% RSLogix 500 project Project6-Final.RSS, saved by version 8.30.00.16 %
PROJECT "UNTITLED"    % processor: Bul.1763 MicroLogix 1100 Series B %

PROGRAM FILES
  LAD 2 "MAIN"  2 rungs
  LAD 3 "LOGIC"  10 rungs

DATA FILES
  O0 OUTPUT  4 elements
  I1 INPUT  6 elements
  S2 STATUS  66 elements
  B3 BINARY  2 elements
  T4 TIMER  1 elements
  C5 COUNTER  4 elements
  R6 CONTROL  1 elements
  N7 INTEGER  4 elements
  F8 FLOAT  1 elements

LADDER 2 "MAIN"
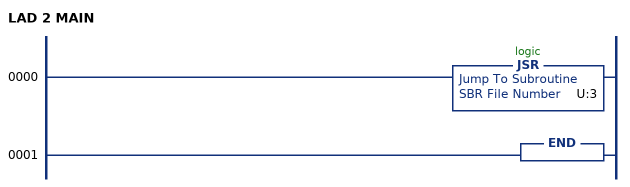
% Rung: 0 %
SOR JSR U:3 EOR
%   U:3  "logic" %
% Rung: 1 %
SOR END EOR

LADDER 3 "LOGIC"
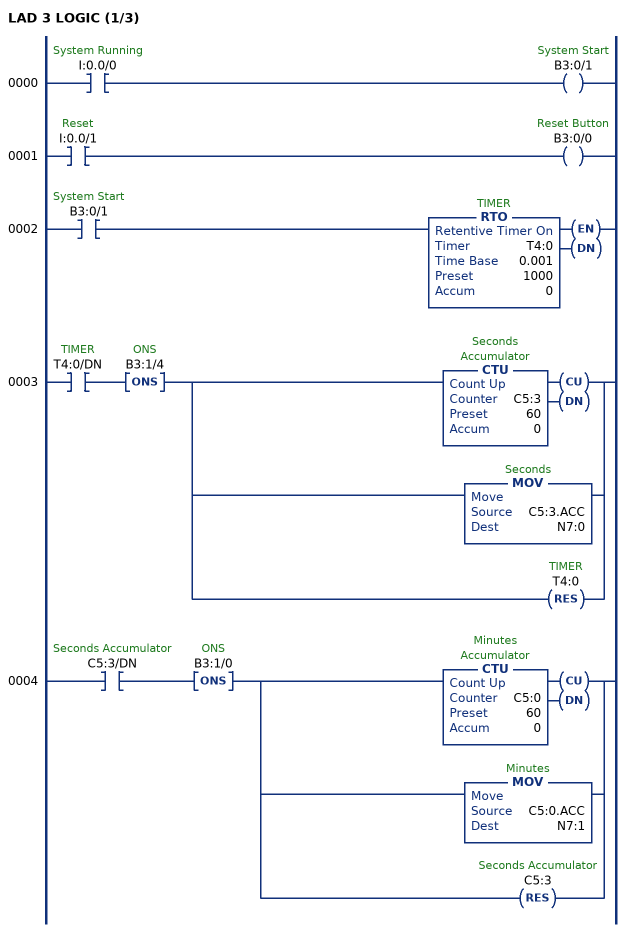
% Rung: 0 %
SOR XIC I:0.0/0 OTE B3:0/1 EOR
%   I:0.0/0  "System Running" %
%   B3:0/1  "System Start" %
% Rung: 1 %
SOR XIC I:0.0/1 OTE B3:0/0 EOR
%   I:0.0/1  "Reset" %
%   B3:0/0  "Reset Button" %
% Rung: 2 %
SOR XIC B3:0/1 RTO T4:0 0.001 1000 0 EOR
%   B3:0/1  "System Start" %
%   T4:0  "TIMER" %
% Rung: 3 %
SOR XIC T4:0/DN ONS B3:1/4 BST CTU C5:3 60 0 NXB MOV C5:3.ACC N7:0 NXB RES T4:0 BND EOR
%   T4:0  "TIMER" %
%   B3:1/4  "ONS" %
%   C5:3  "Seconds Accumulator" %
%   N7:0  "Seconds" %
% Rung: 4 %
SOR XIC C5:3/DN ONS B3:1/0 BST CTU C5:0 60 0 NXB MOV C5:0.ACC N7:1 NXB RES C5:3 BND EOR
%   C5:3  "Seconds Accumulator" %
%   B3:1/0  "ONS" %
%   C5:0  "Minutes Accumulator" %
%   N7:1  "Minutes" %

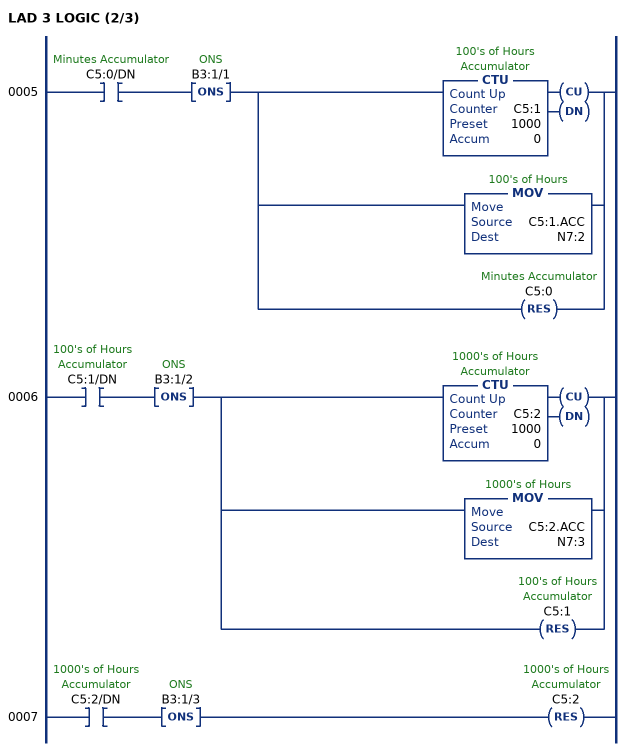
% Rung: 5 %
SOR XIC C5:0/DN ONS B3:1/1 BST CTU C5:1 1000 0 NXB MOV C5:1.ACC N7:2 NXB RES C5:0 BND EOR
%   C5:0  "Minutes Accumulator" %
%   B3:1/1  "ONS" %
%   C5:1  "100's of Hours Accumulator" %
%   N7:2  "100's of Hours" %
% Rung: 6 %
SOR XIC C5:1/DN ONS B3:1/2 BST CTU C5:2 1000 0 NXB MOV C5:2.ACC N7:3 NXB RES C5:1 BND EOR
%   C5:1  "100's of Hours Accumulator" %
%   B3:1/2  "ONS" %
%   C5:2  "1000's of Hours Accumulator" %
%   N7:3  "1000's of Hours" %
% Rung: 7 %
SOR XIC C5:2/DN ONS B3:1/3 RES C5:2 EOR
%   C5:2  "1000's of Hours Accumulator" %
%   B3:1/3  "ONS" %

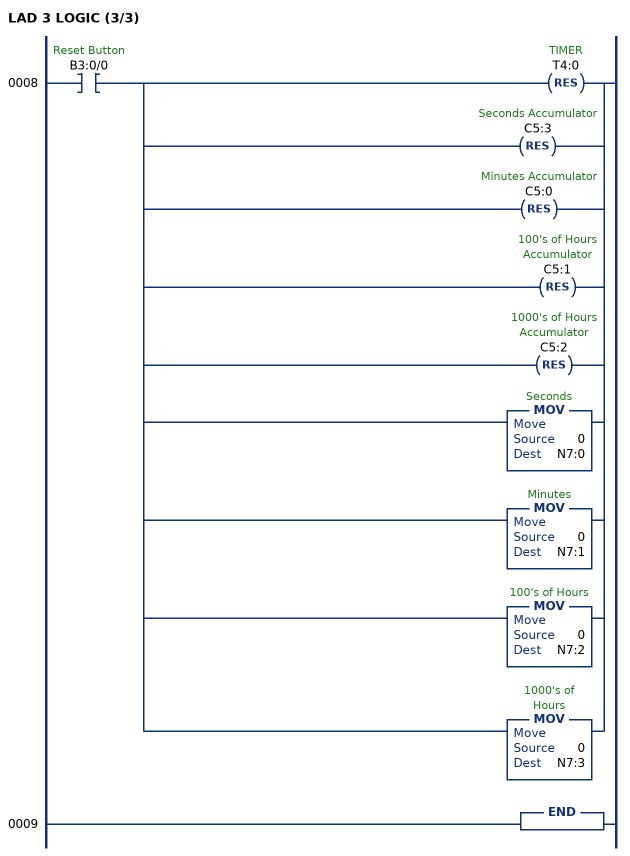
% Rung: 8 %
SOR XIC B3:0/0 BST RES T4:0 NXB RES C5:3 NXB RES C5:0 NXB RES C5:1 NXB RES C5:2 NXB MOV 0 N7:0 NXB MOV 0 N7:1 NXB MOV 0 N7:2 NXB MOV 0 N7:3 BND EOR
%   B3:0/0  "Reset Button" %
%   T4:0  "TIMER" %
%   C5:3  "Seconds Accumulator" %
%   C5:0  "Minutes Accumulator" %
%   C5:1  "100's of Hours Accumulator" %
%   C5:2  "1000's of Hours Accumulator" %
%   N7:0  "Seconds" %
%   N7:1  "Minutes" %
%   N7:2  "100's of Hours" %
%   N7:3  "1000's of Hours" %
% Rung: 9 %
SOR END EOR

DATA TABLE (non-zero values as saved)
DATA T4
% .PRE .ACC %
% T4:0 % 1000 0
DATA C5
% .PRE .ACC %
% C5:0 % 60 0
% C5:1 % 1000 0
% C5:2 % 1000 0
% C5:3 % 60 0
